(* IEC 61131-3 sources: Industry-PLC-LLM/data/PLCBEAD_repo/PLCBEAD_PLCEmbed-main/PLC-BEAD/Source/GEB/MATRIX, 1 file *)

(* ---- MATRIX.ST ---- *)
TYPE
	oscat_arb_0_3               : ARRAY [0..3]    OF BYTE;
END_TYPE

FUNCTION BIT_OF_DWORD : BOOL
	VAR_INPUT
		IN : DWORD;
		N : INT;
	END_VAR

	BIT_OF_DWORD := (SHR(IN,N) AND 16#00000001) > 0;
END_FUNCTION

FUNCTION _BYTE_TO_INT:INT
	VAR_INPUT
		IN :	BYTE;
	END_VAR

	_BYTE_TO_INT := USINT_TO_INT(BYTE_TO_USINT(IN));
END_FUNCTION

FUNCTION BIT_LOAD_B:BYTE
	VAR_INPUT
		IN :	BYTE;
		VAL :	BOOL;
		POS :	INT;
	END_VAR

	IF VAL THEN
		BIT_LOAD_B := IN OR SHL(BYTE#1,POS);
	ELSE
		BIT_LOAD_B := IN AND (NOT SHL(BYTE#1,POS));
	END_IF;
END_FUNCTION

FUNCTION_BLOCK MATRIX_Block

	VAR_INPUT
		X1 :	BOOL;
		X2 :	BOOL;
		X3 :	BOOL;
		X4 :	BOOL;
		X5 :	BOOL;
		RELEASE :	BOOL;
	END_VAR

	VAR_OUTPUT
		CODE :	BYTE;
		_TP :	BOOL;
		Y1 :	BOOL := TRUE;
		Y2 :	BOOL;
		Y3 :	BOOL;
		Y4 :	BOOL;
	END_VAR

	VAR
		line :	BYTE;
		X :	oscat_arb_0_3;
		L :	oscat_arb_0_3;
		i :	INT;
		temp :	BYTE;
		temp2 :	BYTE;
		L_temp :	BYTE;
		temp_bit :	BOOL;
		in_temp :	INT;
	END_VAR

	_TP := FALSE;
	code := BYTE#0;

	(* read scan lines *)
	in_temp := _BYTE_TO_INT(line);
	temp := X[in_temp];  (* X[LINE] umkopieren *)

	temp:=BIT_LOAD_B(temp,X1,0); (* X[line].0 := X1; *)
	temp:=BIT_LOAD_B(temp,X2,1); (* X[line].1 := X2; *)
	temp:=BIT_LOAD_B(temp,X3,2); (* X[line].2 := X3; *)
	temp:=BIT_LOAD_B(temp,X4,3); (* X[line].3 := X4; *)
	temp:=BIT_LOAD_B(temp,X5,4); (* X[line].4 := X5; *)

	X[in_temp] := temp; (* X[LINE] zur�ckkopieren *)

	(* compare for CHAnge *)
	FOR i := 0 TO 3 DO
		IF X[i] <> L[i] THEN
			(* scan line information has CHAnged code need to be found and generated *)
			temp   := x[i] XOR L[i];
			temp2  := X[i];
			L_temp := L[i];

			IF BIT_OF_DWORD(BYTE_TO_DWORD(temp),0) THEN (* temp.X0 *)
				code := BYTE#1;
				temp_bit := BIT_OF_DWORD(BYTE_TO_DWORD(temp2),0);   (* X[i].X0 *)
				code := BIT_LOAD_B(code,temp_bit,7);     			(* code.X7 *)
				L_temp := BIT_LOAD_B(L_temp,temp_bit,0); 			(* L[i].X0 *)
			ELSIF BIT_OF_DWORD(BYTE_TO_DWORD(temp),1) THEN          (* temp.X1 *)
				code := BYTE#2;
				temp_bit := BIT_OF_DWORD(BYTE_TO_DWORD(temp2),1);   (* X[i].X1 *)
				code := BIT_LOAD_B(code,temp_bit,7);     			(* code.X7 *)
				L_temp := BIT_LOAD_B(L_temp,temp_bit,1); 			(* L[i].X1 *)
			ELSIF BIT_OF_DWORD(BYTE_TO_DWORD(temp),2) THEN          (* temp.X2 *)
				code := BYTE#3;
				temp_bit := BIT_OF_DWORD(BYTE_TO_DWORD(temp2),2);   (* X[i].X2 *)
				code := BIT_LOAD_B(code,temp_bit,7);     			(* code.X7 *)
				L_temp := BIT_LOAD_B(L_temp,temp_bit,2); 			(* L[i].X2 *)
			ELSIF BIT_OF_DWORD(BYTE_TO_DWORD(temp),3) THEN          (* temp.X3 *)
				code := BYTE#4;
				temp_bit := BIT_OF_DWORD(BYTE_TO_DWORD(temp2),3);   (* X[i].X3 *)
				code := BIT_LOAD_B(code,temp_bit,7);     			(* code.X7 *)
				L_temp := BIT_LOAD_B(L_temp,temp_bit,3); 			(* L[i].X3 *)
			ELSIF BIT_OF_DWORD(BYTE_TO_DWORD(temp),4) THEN          (* temp.X4 *)
				code := BYTE#5;
				temp_bit := BIT_OF_DWORD(BYTE_TO_DWORD(temp2),4);   (* X[i].X4 *)
				code := BIT_LOAD_B(code,temp_bit,7);     			(* code.X7 *)
				L_temp := BIT_LOAD_B(L_temp,temp_bit,4); 			(* L[i].X4 *)
			END_IF;
			L[i] := L_temp;
			_TP := TRUE;
			code := (code AND BYTE#2#1000_1111) OR SHL(LINE AND BYTE#2#0000_0111,4);
			(* obere zeile enspricht: Code.X4 := Line.X0; /  Code.X5 := Line.X1; / Code.X6 := Line.X2; *)

			(* check if release codes need to be killed *)
			IF NOT release AND code < BYTE#127 THEN
				code := BYTE#0;
				_TP := FALSE;
			END_IF;
			EXIT;
		END_IF;
	END_FOR;

	(* INCrement scan line every cycle *)
	line := INT_TO_BYTE(_BYTE_TO_INT(line) + 1) AND BYTE#2#0000_0011;
	temp := SHL(BYTE#1,_BYTE_TO_INT(line));

	Y1 := BIT_OF_DWORD(BYTE_TO_DWORD(temp),0); (* temp.0 *)
	Y2 := BIT_OF_DWORD(BYTE_TO_DWORD(temp),1); (* temp.1 *)
	Y3 := BIT_OF_DWORD(BYTE_TO_DWORD(temp),2); (* temp.2 *)
	Y4 := BIT_OF_DWORD(BYTE_TO_DWORD(temp),3); (* temp.3 *)

END_FUNCTION_BLOCK

PROGRAM program0

	VAR
		X1 :	BOOL;
		X2 :	BOOL;
		X3 :	BOOL;
		X4 :	BOOL;
		X5 :	BOOL;
		RELEASE :	BOOL;

		CODE :	BYTE;
		_TP :	BOOL;
		Y1 :	BOOL := TRUE;
		Y2 :	BOOL;
		Y3 :	BOOL;
		Y4 :	BOOL;

		func_block : MATRIX_Block;
	END_VAR
	func_block.X1 := X1;
	func_block.X2 := X2;
	func_block.X3 := X3;
	func_block.X4 := X4;
	func_block.X5 := X5;
	func_block.RELEASE := RELEASE;
	func_block();
	CODE := func_block.CODE;
	_TP := func_block._TP;
	Y1 := func_block.Y1;
	Y2 := func_block.Y2;
	Y3 := func_block.Y3;
	Y4 := func_block.Y4;

END_PROGRAM
